PROGRAM MAIN
VAR
	AxisControl : AxisControl;
	sizeMeasure : sizeMeasure;
	weightMeasure : WeightMeasure;
	
END_VAR

AxisControl();
sizeMeasure();
weightMeasure();

//Size in cm
sizeMeasure.sizeInCm;

//Wweight in kg
weightMeasure.weightInKg;

//Breed calculation
BreedCalculation();

//Save new bin position
SaveNewBinPosition();

//Manual motion of servo
ServoManualMotion();

END_PROGRAM

(* stored: Version 1.1.0.1, ProductVersion 3.1.4024.13
   POU MAIN: Id {d7bd07a9-632a-4512-a44e-2ca193c0ff70}, SpecialFunc None *)
